{attribute 'qualified_only'}
VAR_GLOBAL
	//current data being shown
	dataCurrentVisu:structAnalysis;

	data1:structAnalysis;
	data2:structAnalysis;
	data3:structAnalysis;
	
	
END_VAR

(* stored: Version 1.1.0.1, ProductVersion 3.1.4024.11
   GVL dataGrab: Id {c4f9d33c-8c0c-018b-158e-5709296def3f} *)
